# EPICS autosave request: iocBoot/bkhDigiI.req
$(P):BI:$(MOD):BIT$(N).DESC
$(P):BI:$(MOD):BIT$(N).VAL
